FUNCTION_BLOCK Section4Ctrl (* Basic Function Block Type *)
  (* Standard: 61499-2 *)
  (* Version 0.0, 5/27/2018, MIA, nxtControl GmbH, Template *)
  PACKAGE Main;
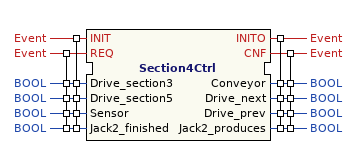
  EVENT_INPUT
    INIT WITH Drive_section3, Drive_section5, Sensor, Jack2_finished; (* Initialization Request *)
    REQ WITH Drive_section3, Drive_section5, Sensor, Jack2_finished; (* Normal Execution Request *)
  END_EVENT
  EVENT_OUTPUT
    INITO WITH Conveyor, Drive_next, Drive_prev, Jack2_produces; (* Initialization Confirm *)
    CNF WITH Conveyor, Drive_next, Drive_prev, Jack2_produces; (* Execution Confirmation *)
  END_EVENT
  VAR_INPUT
    Drive_section3 : BOOL; (* Input event qualifier *)
    Drive_section5 : BOOL;
    Sensor : BOOL;
    Jack2_finished : BOOL;
  END_VAR
  VAR_OUTPUT
    Conveyor : BOOL; (* Output event qualifier *)
    Drive_next : BOOL;
    Drive_prev : BOOL;
    Jack2_produces : BOOL;
  END_VAR
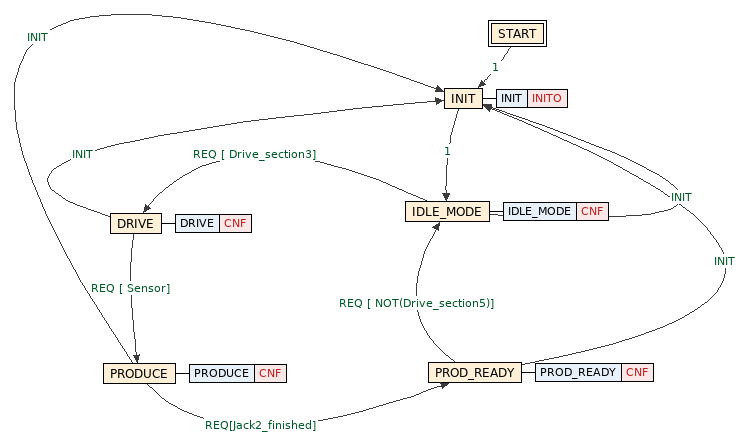
  EC_STATES
    START; (* Initial State *)
    INIT : INIT -> INITO; (* Initialization *)
    IDLE_MODE : IDLE_MODE -> CNF;
    DRIVE : DRIVE -> CNF;
    PRODUCE : PRODUCE -> CNF;
    PROD_READY : PROD_READY -> CNF;
  END_STATES
  EC_TRANSITIONS
    START TO INIT := 1;
    INIT TO IDLE_MODE := 1;
    IDLE_MODE TO DRIVE := REQ [ Drive_section3];
    DRIVE TO PRODUCE := REQ [ Sensor];
    PRODUCE TO PROD_READY := REQ[Jack2_finished];
    PROD_READY TO IDLE_MODE := REQ [ NOT(Drive_section5)];
    DRIVE TO INIT := INIT;
    IDLE_MODE TO INIT := INIT;
    PROD_READY TO INIT := INIT;
    PRODUCE TO INIT := INIT;
  END_TRANSITIONS
  ALGORITHM INIT IN ST: (* Initialization algorithm *)
;
Conveyor := FALSE;
Jack2_produces := FALSE;
Drive_prev := FALSE;
Drive_next := FALSE;
  END_ALGORITHM
  ALGORITHM IDLE_MODE IN ST:
Conveyor := FALSE;
Jack2_produces := FALSE;
Drive_prev := TRUE;
Drive_next := FALSE;
  END_ALGORITHM
  ALGORITHM DRIVE IN ST:
Conveyor := TRUE;
Jack2_produces := FALSE;
Drive_prev := TRUE;
Drive_next := FALSE;
  END_ALGORITHM
  ALGORITHM PRODUCE IN ST:
Conveyor := FALSE;
Jack2_produces := TRUE;
Drive_prev := FALSE;
Drive_next := FALSE;
  END_ALGORITHM
  ALGORITHM PROD_READY IN ST:
Conveyor := TRUE;
Jack2_produces := FALSE;
Drive_prev := TRUE;
Drive_next := TRUE;
  END_ALGORITHM
END_FUNCTION_BLOCK
